ABB RobotStudio station: assignment1.rsstn

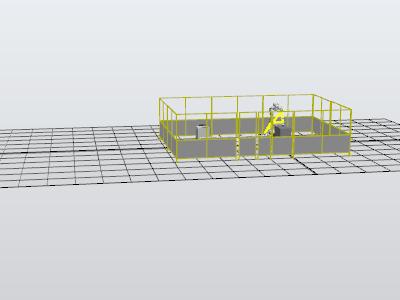
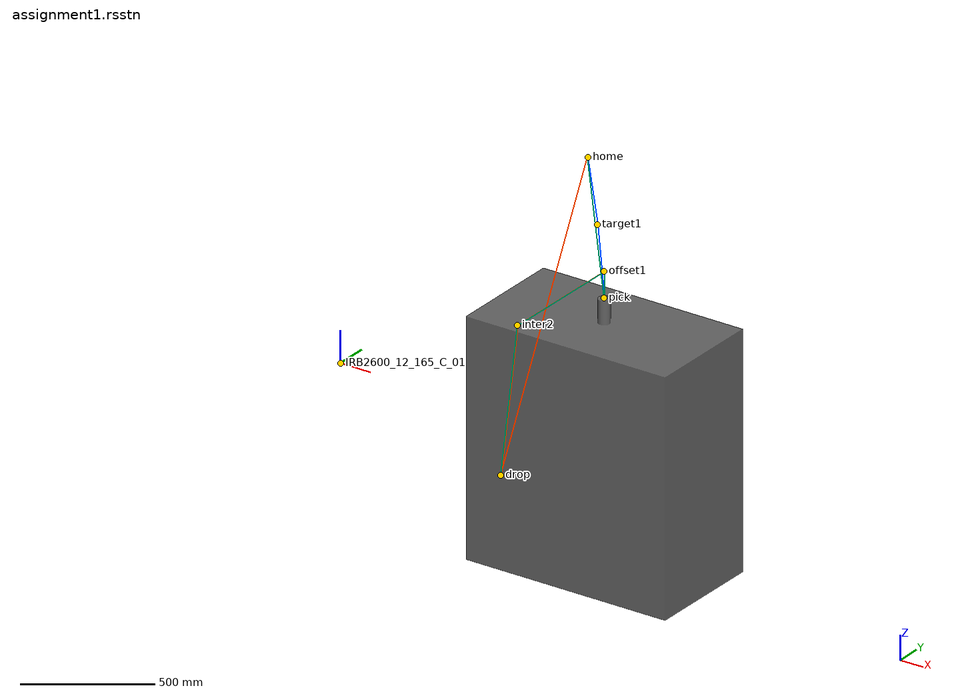
[picture v1: parts stored in the station drawn from their meshes, with robot base, taught points and paths (robot models come from the ABB library and are not in the file)]
Station Station (saved by RobotStudio 22.3.10141.1)
Controller Controller6, task T_ROB1: task frame (RAPID world) sits at (0, 0, 542.78) mm in the station
Controller Controller6
  mechanical unit ROB_1: IRB2600_12_165_C_01, 6 joints, base frame (0, 0, 0) mm
Layout (positions relative to the parent item):
  - concrate [part, from Libraries\concrate.rslib] at (-450, -450, 0) mm
  - Robotpedestal1400_H240 [part, from Equipment\Robot Pedestal 1400 H240.rslib] at (-30, 0, 302.67) mm
  - IRB2600_12_165_C_01 [mechanism, from %ABB.RobotStudio.Models.IRB2600%\IRB2600_12_165_C_01.rslib] at (0, 0, 542.78) mm; joint values [0, 0, 0, 0, 0.5236, 0] (rad or m)
  - 400_guide [part, from Equipment\Conveyor Guide 400.rslib] at (936.98, -557.07, -194.19) mm, rotated rx 1.7 ry 0.02 rz -90.65 deg
  - IRC5_Control-Module [part, from Equipment\IRC5_Control-Module.rslib] at (-1446.28, -2888.11, 100) mm, rotated rx 90 ry 0 rz 178.48 deg
  - Part_1 [part] at (690.39, -177.58, 0) mm, size 900 x 500 x 1000 mm
  - Part_2 [part] at (1140.39, 72.42, 1000) mm, size 50 x 49.9 x 100 mm
  - SmartComponent_3 [smart component] at (1018.61, 0, 1760.28) mm, rotated rx 180 ry 60 rz 180 deg
      signals: DI atacher
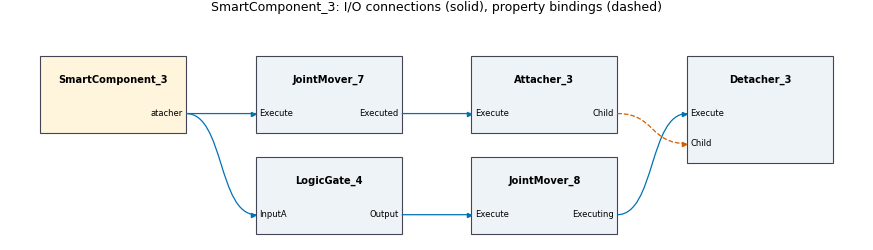
      connections:
        SmartComponent_3.atacher -> JointMover_7.Execute
        JointMover_7.Executed -> Attacher_3.Execute
        JointMover_8.Executing -> Detacher_3.Execute
        LogicGate_4.Output -> JointMover_8.Execute
        SmartComponent_3.atacher -> LogicGate_4.InputA
        Attacher_3.Child => Detacher_3.Child
    - JointMover_7 [smart component, from Components\JointMover.rslib]
        properties: Mechanism=Smart_Gripper_Servo_Fingers_2; Relative=false; Duration=0; J1=0.024
    - JointMover_8 [smart component, from Components\JointMover.rslib]
        properties: Mechanism=Smart_Gripper_Servo_Fingers_2; Relative=false; Duration=0; J1=0.025
    - Attacher_3 [smart component, from Components\Attacher.rslib]
        properties: Parent=Smart_Gripper_Servo_Fingers_2; Flange=0; Child=Part_2; Mount=false; Offset=[0 0 0]; Orientation=[0 0 0]
    - LogicGate_4 [smart component, from Components\LogicGate.rslib]
        properties: Operator=NOT; Delay=0
    - Detacher_3 [smart component, from Components\Detacher.rslib]
        properties: Child=Part_2; KeepPosition=true
    - Smart_Gripper_Servo_Fingers_2 [mechanism, from Tools\ABB_Smart_Gripper_Servo_Fingers.rslib] at (0, 0, 0) mm; joint values [0.025] (rad or m)
  - Fence_2500 [graphiccomponentgroup, from Equipment\Fence_2500.rslib] at (-2001.06, 0, 0) mm
    - Body 1 [part, from Equipment\Fence_2500.rslib]
    - Body 2 [part, from Equipment\Fence_2500.rslib]
  - Fence_2500_2 [graphiccomponentgroup, from Equipment\Fence_2500.rslib] at (-1994.36, -2494.92, 0) mm
    - Body 1 [part, from Equipment\Fence_2500.rslib]
    - Body 2 [part, from Equipment\Fence_2500.rslib]
  - Fence_2500_3 [graphiccomponentgroup, from Equipment\Fence_2500.rslib] at (-1975.9, -4986.56, 0) mm
    - Body 1 [part, from Equipment\Fence_2500.rslib]
    - Body 2 [part, from Equipment\Fence_2500.rslib]
  - Fence_2500_4 [graphiccomponentgroup, from Equipment\Fence_2500.rslib] at (492.5, 2452.07, 0) mm, rotated rx 0 ry 0 rz 89.22 deg
    - Body 1 [part, from Equipment\Fence_2500.rslib]
    - Body 2 [part, from Equipment\Fence_2500.rslib]
  - Fence_2500_5 [graphiccomponentgroup, from Equipment\Fence_2500.rslib] at (564.17, 2477.21, 7.49) mm, rotated rx 0 ry 0 rz -90.99 deg
    - Body 1 [part, from Equipment\Fence_2500.rslib]
    - Body 2 [part, from Equipment\Fence_2500.rslib]
  - Fence_2500_6 [graphiccomponentgroup, from Equipment\Fence_2500.rslib] at (-1994.53, -4973.46, -10.64) mm, rotated rx 0 ry 0 rz -89.38 deg
    - Body 1 [part, from Equipment\Fence_2500.rslib]
    - Body 2 [part, from Equipment\Fence_2500.rslib]
  - Fence_2500_8 [graphiccomponentgroup, from Equipment\Fence_2500.rslib] at (514.73, -4940.61, -13.4) mm, rotated rx 0 ry 0 rz -89.19 deg
    - Body 1 [part, from Equipment\Fence_2500.rslib]
    - Body 2 [part, from Equipment\Fence_2500.rslib]
  - Fence_2500_9 [graphiccomponentgroup, from Equipment\Fence_2500.rslib] at (3065.79, -17.39, 0) mm
    - Body 1 [part, from Equipment\Fence_2500.rslib]
    - Body 2 [part, from Equipment\Fence_2500.rslib]
  - Fence_2500_10 [graphiccomponentgroup, from Equipment\Fence_2500.rslib] at (3071.96, -4918.94, 0) mm
    - Body 1 [part, from Equipment\Fence_2500.rslib]
    - Body 2 [part, from Equipment\Fence_2500.rslib]
  - Gate_3 [graphiccomponentgroup, from Equipment\Fence_Gate.rslib] at (3057.19, -1532.75, 0) mm
    - Body 1 [part, from Equipment\Fence_Gate.rslib]
    - Body 2 [part, from Equipment\Fence_Gate.rslib]
    - Body 3 [part, from Equipment\Fence_Gate.rslib]
  - Fence_740 [graphiccomponentgroup, from Equipment\Fence_740.rslib] at (3028.18, -2317.96, 0) mm
    - Body 1 [part, from Equipment\Fence_740.rslib]
    - Body 2 [part, from Equipment\Fence_740.rslib]
Attachment: SmartComponent_3 is attached to IRB2600_12_165_C_01 / Link6
Station logic (signal -> signal, property => property):
  Controller6.atach -> SmartComponent_3.atacher
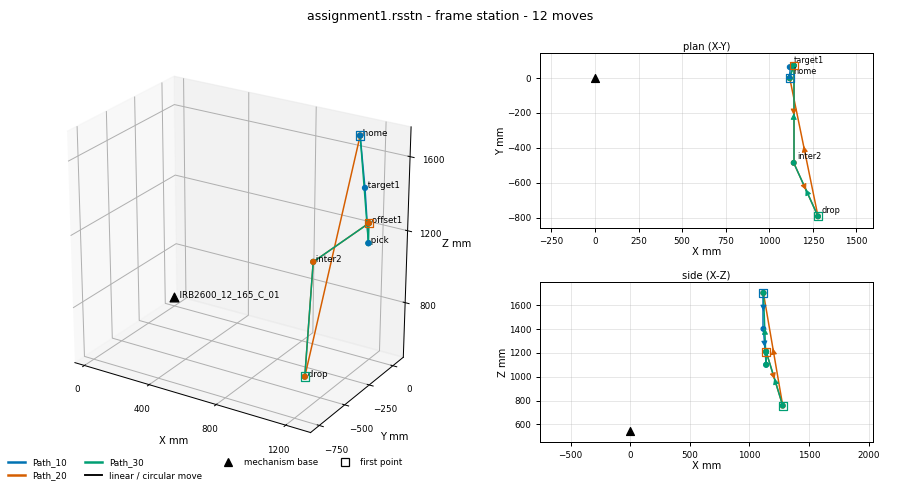
[picture p0: tool path of assignment1.rsstn in frame station, 12 of 12 moves have a stored position in this frame; points joined in program order, loops and branches not executed]
Targets, tools, work objects and paths stored in the station, written as RAPID:
! task T_ROB1
MODULE CalibData
  PERS tooldata Servo:=[TRUE,[[0,0,114.2],[1,0,0,0]],[0.215,[8.7,12.3,49.2],[1,0,0,0],0.00021,0.00024,0.00009]];
ENDMODULE

! task T_ROB1
MODULE Module1
  CONST robtarget home:=[[1117.512260434,0,1160.4],[0.5,0,0.866025404,0],[0,0,0,0],[9E+09,9E+09,9E+09,9E+09,9E+09,9E+09]];
  CONST robtarget target1:=[[1117.51196729,63.415861744,858.74614082],[0.500000011,-0.00000001,0.866025397,-0.000000006],[0,-1,0,0],[9E+09,9E+09,9E+09,9E+09,9E+09,9E+09]];
  CONST robtarget pick:=[[1140.393001636,72.422767793,557.216016575],[0.014410605,-0.000000016,0.999896162,0.000000003],[0,-1,0,0],[9E+09,9E+09,9E+09,9E+09,9E+09,9E+09]];
  CONST robtarget offset1:=[[1140.393016467,72.422768952,667.788108044],[0.014410635,-0.000000015,0.999896161,0.000000005],[0,-1,0,0],[9E+09,9E+09,9E+09,9E+09,9E+09,9E+09]];
  CONST robtarget inter2:=[[1140.39300548,-486.040786199,667.788126074],[0.014410639,-0.000000029,0.999896161,0],[-1,0,-1,0],[9E+09,9E+09,9E+09,9E+09,9E+09,9E+09]];
  CONST robtarget drop:=[[1279.7280634,-793.096378817,214.208572534],[0.014410588,-0.000000067,0.999896162,0.000000007],[-1,0,-1,0],[9E+09,9E+09,9E+09,9E+09,9E+09,9E+09]];
  PROC Path_10()
    MoveL home,v1000,z100,Servo\WObj:=wobj0;
    MoveL target1,v1000,z100,Servo\WObj:=wobj0;
    MoveL pick,v1000,z100,Servo\WObj:=wobj0;
    WaitTime 1;
    SetDO atach,1;
  ENDPROC
  PROC Path_20()
    MoveL offset1,v1000,z100,Servo\WObj:=wobj0;
    MoveL inter2,v1000,z100,Servo\WObj:=wobj0;
    MoveL drop,v1000,z100,Servo\WObj:=wobj0;
    WaitTime 1;
    SetDO atach,0;
    MoveL home,v1000,z100,Servo\WObj:=wobj0;
  ENDPROC
  PROC Path_30()
    MoveL drop,v1000,z100,Servo\WObj:=wobj0;
    WaitTime 1;
    SetDO atach,1;
    MoveL inter2,v1000,z100,Servo\WObj:=wobj0;
    MoveL offset1,v1000,z100,Servo\WObj:=wobj0;
    MoveL pick,v1000,z100,Servo\WObj:=wobj0;
    WaitTime 1;
    SetDO atach,0;
    MoveL home,v1000,z100,Servo\WObj:=wobj0;
  ENDPROC
  PROC Path_40()
    Path_10;
    Path_20;
    Path_30;
  ENDPROC
ENDMODULE

